{attribute 'GeneratedUsingTerminal: EJ3318-0000-0017'}
{attribute addProperty BoxType "EJ3318-0000-0017"}
{attribute addProperty Id "TC_Channel_1AT %I*TC_Channel_9575FEA17TC_Channel_2AT %I*TC_Channel_9575FEA17TC_Channel_3AT %I*TC_Channel_9575FEA17TC_Channel_4AT %I*TC_Channel_9575FEA17TC_Channel_5AT %I*TC_Channel_9575FEA17TC_Channel_6AT %I*TC_Channel_9575FEA17TC_Channel_7AT %I*TC_Channel_9575FEA17TC_Channel_8AT %I*TC_Channel_9575FEA17RTD_Inputs_Channel_1AT %I*RTD_Inputs_Channel_9575FEA17RTD_Inputs_Channel_2AT %I*RTD_Inputs_Channel_9575FEA17WcStateAT %I*WcState_9091E0EB2InfoDataAT %I*InfoData_94A18F5E2"}
{attribute addProperty CRC "2421106243"}
{attribute addProperty Size "74"}
TYPE EJ3318_904F2643 EXTENDS EtcSlaveTerminalBase_947E5A46 :
STRUCT
	{attribute addProperty Name "TC_Channel_1"}
	TC_Channel_1 : TC_Channel_9575FEA1;
	{attribute addProperty Name "TC_Channel_2"}
	TC_Channel_2 : TC_Channel_9575FEA1;
	{attribute addProperty Name "TC_Channel_3"}
	TC_Channel_3 : TC_Channel_9575FEA1;
	{attribute addProperty Name "TC_Channel_4"}
	TC_Channel_4 : TC_Channel_9575FEA1;
	{attribute addProperty Name "TC_Channel_5"}
	TC_Channel_5 : TC_Channel_9575FEA1;
	{attribute addProperty Name "TC_Channel_6"}
	TC_Channel_6 : TC_Channel_9575FEA1;
	{attribute addProperty Name "TC_Channel_7"}
	TC_Channel_7 : TC_Channel_9575FEA1;
	{attribute addProperty Name "TC_Channel_8"}
	TC_Channel_8 : TC_Channel_9575FEA1;
	{attribute addProperty Name "RTD_Inputs_Channel_1"}
	RTD_Inputs_Channel_1 : RTD_Inputs_Channel_9575FEA1;
	{attribute addProperty Name "RTD_Inputs_Channel_2"}
	RTD_Inputs_Channel_2 : RTD_Inputs_Channel_9575FEA1;
	{attribute addProperty Name "WcState"}
	WcState : WcState_9091E0EB;
	{attribute addProperty Name "InfoData"}
	InfoData : InfoData_94A18F5E;
END_STRUCT
END_TYPE

(* stored: Version 1.2.0.0, ProductVersion 3.1.4024.9
   DUT EJ3318_904F2643: Id {818f5917-f9f6-429e-bd80-1893bfdf34fe} *)
